{attribute addProperty BoxType "EL2258-0000-0017"}
{attribute addProperty Id "MTO_Inputs_ChannelAT %I*ARRAY[0..7] OF MTO_Inputs_Channel_5AD475AF8721090MTO_Outputs_10x_ChannelAT %Q*ARRAY[0..7] OF MTO_Outputs_10x_Channel_24D255B145285660WcStateAT %I*WcState_F855686C1620InfoDataAT %I*InfoData_0BDED7BF144180"}
{attribute addProperty CRC "2477755315"}
{attribute addProperty SizeInBites "5560"}
{attribute addProperty SizeInBytes "695"}
TYPE EL2258_5305AE3B :
STRUCT
	{attribute addProperty Name "MTO_Inputs_Channel"}
	MTO_Inputs_Channel : ARRAY[0..7] OF MTO_Inputs_Channel_5AD475AF;
	{attribute addProperty Name "MTO_Outputs_10x_Channel"}
	MTO_Outputs_10x_Channel : ARRAY[0..7] OF MTO_Outputs_10x_Channel_24D255B1;
	{attribute addProperty Name "WcState"}
	WcState : WcState_F855686C;
	{attribute addProperty Name "InfoData"}
	InfoData : InfoData_0BDED7BF;
END_STRUCT
END_TYPE

(* stored: Version 1.2.0.0, ProductVersion 3.1.4024.9
   DUT EL2258_5305AE3B: Id {3b24f661-8eab-4c5c-b90f-5c78948b8845} *)
